// TIA Portal V20 export
// export: Created 2025-12-01T14:56:19.2434616Z, ExportSetting None, DisplayName Totally Integrated Automation Portal, DisplayVersion V20 Update 3, DisplayName TIA Portal Openness, DisplayVersion V20 Update 3, DisplayName TIA Portal Version Control Interface, DisplayVersion V20 Update 3, DisplayName STEP 7 Professional, DisplayVersion V20 Update 3, DisplayName STEP 7 Safety, DisplayVersion V20 Update 2, DisplayName WinCC Basic/Comfort/Advanced, DisplayVersion V20 Update 3, DisplayName WinCC Professional, DisplayVersion V20 Update 3, DisplayName WinCC Unified, DisplayVersion V20 Update 3
TYPE "i950 Palabra de Control"
   STRUCT
      "Control Signal Bit 0" : Bool;
      "Control Signal Bit 1" : Bool;
      "Activate Quickstop Application" : Bool;
      "Enable Operation" : Bool;
      "Control Signal Bit 4" : Bool;
      "Jog Positive" : Bool;
      "Jog Negative" : Bool;
      "Fault Reset" : Bool;
      Halt : Bool;
      "Execute Homing" : Bool;
      "Home Position Reset" : Bool;
      Abort : Bool;
      "Control Signal Bit 12" : Bool;
      "Activate Vel Override" : Bool;
      "Release Brake Manual" : Bool;
      "Control Signal Bit 15" : Bool;
      Release_Brake : Bool;
      "Profile No 01" : Bool;
      "Profile No 02" : Bool;
      "Profile No 04" : Bool;
      "Profile No 08" : Bool;
      "Execute Positioning" : Bool;
      "Control Signal Bit 21" : Bool;
      "Finish Positioning" : Bool;
      "Disable Toucj Probe" : Bool;
      "Control Signal Bit 24" : Bool;
      "Control Signal Bit 25" : Bool;
      "Control Signal Bit 26" : Bool;
      "Control Signal Bit 27" : Bool;
      "Activate Ext. Position" : Bool;
      "Activate Ext. Velocity" : Bool;
      "Activate Ext. Acc Dec Jerk" : Bool;
      "Activate Ext. Torque Limit" : Bool;
   END_STRUCT;
END_TYPE
